INTERFACE I_Extensions

METHOD PUBLIC Accept
VAR_INPUT
	Visitor : I_ExtensionVisitor;
END_VAR
END_METHOD

METHOD AddExtension
VAR_INPUT
	Extension : I_Extension;
END_VAR
END_METHOD

METHOD PUBLIC TryGetExtensionByName : BOOL
VAR_INPUT
	Name : T_MAXSTRING;
	Destination : REFERENCE TO I_Extension;
END_VAR
END_METHOD

END_INTERFACE

(* stored: Version 1.1.0.1, ProductVersion 3.1.4024.12
   Itf I_Extensions: Id {dddd2dfd-696b-4620-a8f1-aee32e996020}
   Method Accept: Id {6aa6bb47-2e9a-4ee0-b4d4-786587961113}
   Method AddExtension: Id {a44f1c4a-9213-473e-aa2d-d4c8de85f9ba}
   Method TryGetExtensionByName: Id {f35ea915-7d96-4e05-896c-58c994858579} *)
